{attribute 'qualified_only'}
{attribute 'strict'}
TYPE E_Result :
(
	done,
	timeout,
	error,
	interrupt,
	stop
);
END_TYPE

(* stored: Version 1.1.0.1, ProductVersion 3.1.4024.11
   EnumerationTextList E_Result: Id {f75cc079-29a3-4d27-b294-c8ee80cfa1af} *)
